// TIA Portal V17 export
// export: Created 2023-02-23T17:16:27.9480858Z, ExportSetting WithDefaults, DisplayName Totally Integrated Automation Portal, DisplayVersion V17, DisplayName TIA Portal Openness, DisplayVersion V17, DisplayName TIA Portal Version Control Interface, DisplayVersion V17, DisplayName TIA Portal Test Suite Advanced, DisplayVersion V17, DisplayName STEP 7 Professional, DisplayVersion V17, DisplayName SIMATIC Energy Suite, DisplayVersion V17, DisplayName STEP 7 Safety, DisplayVersion V17, DisplayName WinCC Professional, DisplayVersion V17
FUNCTION "MAN_ClassManagement" : Void   // FC3, LAD
{ S7_Optimized_Access := 'TRUE' }
VERSION : 0.1
// stored: AutoNumber true, IsIECCheckEnabled false, SetENOAutomatically false, UDAEnableTagReadback false
BEGIN

REGION Network 1: Call: ChooseMode
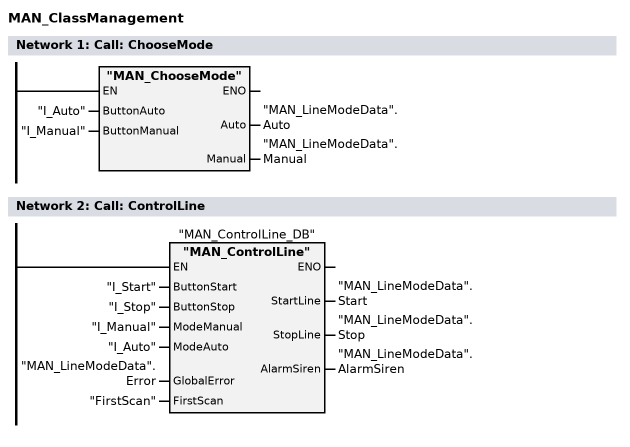
   RUNG wire#powerrail
      "MAN_ChooseMode"(ButtonAuto := "I_Auto", ButtonManual := "I_Manual", Auto => "MAN_LineModeData".Auto, Manual => "MAN_LineModeData".Manual)
   END_RUNG
   // the same network as SCL:
   "MAN_ChooseMode"(ButtonAuto := "I_Auto",
                    ButtonManual := "I_Manual",
                    Auto => "MAN_LineModeData".Auto,
                    Manual => "MAN_LineModeData".Manual);
END_REGION

REGION Network 2: Call: ControlLine
   RUNG wire#powerrail
      "MAN_ControlLine_DB"(ButtonStart := "I_Start", ButtonStop := "I_Stop", ModeManual := "I_Manual", ModeAuto := "I_Auto", GlobalError := "MAN_LineModeData".Error, FirstScan := "FirstScan", StartLine => "MAN_LineModeData".Start, StopLine => "MAN_LineModeData".Stop, AlarmSiren => "MAN_LineModeData".AlarmSiren)
   END_RUNG
   // the same network as SCL:
   "MAN_ControlLine_DB"(ButtonStart := "I_Start",   // "MAN_ControlLine"
                        ButtonStop := "I_Stop",
                        ModeManual := "I_Manual",
                        ModeAuto := "I_Auto",
                        GlobalError := "MAN_LineModeData".Error,
                        FirstScan := "FirstScan",
                        StartLine => "MAN_LineModeData".Start,
                        StopLine => "MAN_LineModeData".Stop,
                        AlarmSiren => "MAN_LineModeData".AlarmSiren);
END_REGION
END_FUNCTION
